FUNCTION "_getEdges" : Void
TITLE = {"version":"v1.0","author":"cyanezf","family":"core/util","status":"current","deprecatedBy": null,"dependencies" : []}
{ S7_Optimized_Access := 'TRUE' }
AUTHOR : cyanezf
FAMILY : 'core/util'
NAME : _getEdges
VERSION : 1.0

   VAR_INPUT
      bit : Bool;   // Bit to check
   END_VAR

   VAR_OUTPUT
      pulseOn : Bool;   // 1=Bit changes to true
      pulseOff : Bool;   // 1=Bit changes to false
   END_VAR

   VAR_IN_OUT
      fp : Bool;   // IOX: Auxiliary static bit (Not temp bit!)
   END_VAR

BEGIN
(*--
# Documentation

## Log

| version | date | author | description |
|:-------:|:----:|:------:|:------------|
| v1.0 | 2025-03-24 | cyanezf | First version |

## Description

This function returns the positive and negative edges from `bit`.

--*)

	#pulseOn := #bit AND NOT #fp;
	#pulseOff := NOT #bit AND #fp;
	#fp := #bit;
	ENO := true;

END_FUNCTION

